(* CODESYS project tt_serialcommunication.library
   Company: Trimech Technology
   Version: 1.0
   Placeholder: TT_SerialCom_Lib
   Author: Beckhoff Singapore
   Title: TT_SerialCom_Lib

Project tree, tasks and I/O mapping:
  libraries: Tc2_SerialCom, * (Beckhoff Automation GmbH); Tc2_Standard, * (Beckhoff Automation GmbH); Tc2_System, * (Beckhoff Automation GmbH); Tc3_Module, * (Beckhoff Automation GmbH); Tc3_Interfaces, * (Beckhoff Automation GmbH)
  GVL/
    global variables TT_SerialComm_GVL
  Custom Datatypes/
    data type TT_Serial_COMBUFFER
    data type TT_Serial_FunctionResult
    data type TT_Serial_StringFormat
  Version/
    global variables Global_Version
  function block TT_Serial_StandardTask [ST]: ReadString80, SendString80
  function block TT_Serial_FastBackgroundTask [ST]: Update_Channel
  global variables TT_SerialComm_Parameters
*)

// Custom Datatypes/TT_Serial_COMBUFFER
TYPE TT_Serial_COMBUFFER :
STRUCT
(**)
	(* PLC to IO interface *)
	txBuffer 		: ComBuffer;
	rxBuffer 		: ComBuffer;
(**)
(**)	
	(* Buffers for EL COM *)
	rxElComBuffer AT %I* 	: EL6inData22B;
	txElComBuffer AT %Q* 	: EL6outData22B;
(**)
(**)
	(* Buffers for PC COM *)
	rxPcComBuffer AT %I* 	: PcComInData;
	txPcComBuffer AT %Q* 	: PcComOutData;
(**)
END_STRUCT
END_TYPE

// Custom Datatypes/TT_Serial_FunctionResult
TYPE TT_Serial_FunctionResult :
(
	NO_ERROR := -1,
	BUSY := 0,
	COM_SEND_ERROR,
	COM_RECEIVE_ERROR,
	COM_NO_STRING_RECEIVED
);
END_TYPE

// Custom Datatypes/TT_Serial_StringFormat
TYPE TT_Serial_StringFormat :
STRUCT
	Prefix : STRING;
	Surfix : STRING;
END_STRUCT
END_TYPE

// GVL/TT_SerialComm_GVL
VAR_GLOBAL
	SerialComBuffer 	: ARRAY [1..MAX_CHANNELS] OF TT_Serial_ComBuffer;
	SerialStringFormat	: ARRAY [1..MAX_CHANNELS] OF TT_Serial_StringFormat;
END_VAR

// Version/Global_Version
// This function has been automatically generated from the project information.
VAR_GLOBAL CONSTANT
	{attribute 'const_non_replaced'}
	stLibVersion_TT_SerialCom_Lib : ST_LibVersion := (iMajor := 1, iMinor := 0, iBuild := 0, iRevision := 0, sVersion := '1.0');
END_VAR

// TT_SerialComm_Parameters
VAR_GLOBAL CONSTANT
	MAX_CHANNELS 	: INT := 2;
END_VAR

// TT_Serial_StandardTask
FUNCTION_BLOCK TT_Serial_StandardTask
VAR_OUTPUT
END_VAR
VAR
	fbSendString 	: ARRAY[1..MAX_CHANNELS] OF SendString;
	fbReceiveString : ARRAY[1..MAX_CHANNELS] OF ReceiveString; (*String default 80. for 255, use ReceiveString255*)
	
	SendFlag 		: ARRAY[1..MAX_CHANNELS] OF BOOL;
	SendDataBuffer	: ARRAY[1..MAX_CHANNELS] OF STRING;
END_VAR

;

METHOD PUBLIC ReadString80 : TT_Serial_FunctionResult
VAR_INPUT
	CHANNEL 			: INT;
	RECEIVED_DATA		: POINTER TO STRING;
END_VAR
VAR 
	String_Data_Buffer 	: STRING;
END_VAR
fbReceiveString[CHANNEL](
	Prefix:= SerialStringFormat[CHANNEL].Prefix, 
	Suffix:= SerialStringFormat[CHANNEL].Surfix, 
	Timeout:= T#1S, 
	ReceivedString:= String_Data_Buffer, 
	RXbuffer:= SerialComBuffer[CHANNEL].rxBuffer );
IF fbReceiveString[CHANNEL].Error > 0 THEN
	ReadString80 := TT_Serial_FunctionResult.COM_RECEIVE_ERROR;
END_IF
IF fbReceiveString[CHANNEL].StringReceived THEN
	RECEIVED_DATA^ := String_Data_Buffer;
	ReadString80 := TT_Serial_FunctionResult.NO_ERROR;
ELSIF fbReceiveString[CHANNEL].Busy THEN
	ReadString80 := TT_Serial_FunctionResult.BUSY;
ELSE
	ReadString80 := TT_Serial_FunctionResult.COM_NO_STRING_RECEIVED;
END_IF
END_METHOD

METHOD PUBLIC SendString80 : TT_Serial_FunctionResult
VAR_INPUT
	CHANNEL	: INT;		(* The Serial Comm channel to send *)
	DATA	: STRING;	(* Without prefix & surfix *)
END_VAR
VAR
	fbTRIG 	: F_TRIG;
END_VAR
SendDataBuffer[CHANNEL] := CONCAT(SerialStringFormat[CHANNEL].Prefix, CONCAT(DATA, SerialStringFormat[CHANNEL].Surfix));
fbSendString[CHANNEL](SendString:= SendDataBuffer[CHANNEL], TXbuffer:= SerialComBuffer[CHANNEL].txBuffer);
IF fbSendString[CHANNEL].Error > 0 THEN
	SendString80 := TT_Serial_FunctionResult.COM_SEND_ERROR;
END_IF
IF fbSendString[CHANNEL].Busy THEN
	SendString80 := TT_Serial_FunctionResult.BUSY;
ELSE
	SendString80 := TT_Serial_FunctionResult.NO_ERROR;
END_IF
END_METHOD

END_FUNCTION_BLOCK

// TT_Serial_FastBackgroundTask
FUNCTION_BLOCK TT_Serial_FastBackgroundTask
VAR
	fbSerialLineControl	: ARRAY[1..MAX_CHANNELS] OF SERIALLINECONTROL;
END_VAR

;

METHOD PUBLIC Update_Channel : INT
VAR_INPUT
	CHANNEL : INT;
END_VAR
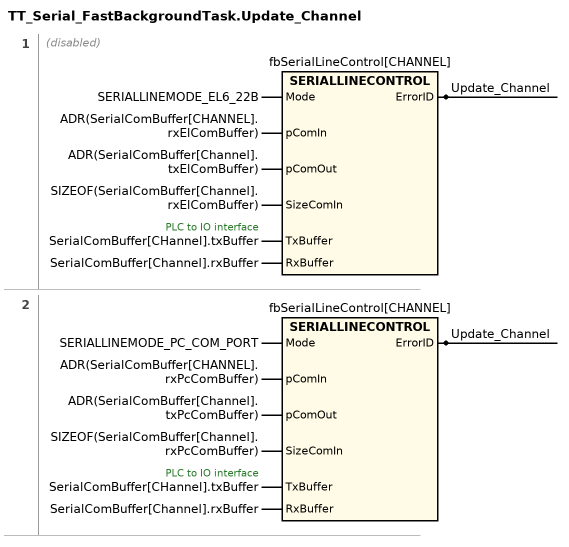
// NETWORK 1 (disabled)
//   SerialComBuffer[CHannel].txBuffer: PLC to IO interface
// fbSerialLineControl[CHANNEL](
//     Mode := SERIALLINEMODE_EL6_22B,
//     pComIn := ADR(SerialComBuffer[CHANNEL].rxElComBuffer),
//     pComOut := ADR(SerialComBuffer[Channel].txElComBuffer),
//     SizeComIn := SIZEOF(SerialComBuffer[Channel].rxElComBuffer),
//     TxBuffer := SerialComBuffer[CHannel].txBuffer,
//     RxBuffer := SerialComBuffer[Channel].rxBuffer,
//     ErrorID => Update_Channel); // SERIALLINECONTROL

// NETWORK 2
//   SerialComBuffer[CHannel].txBuffer: PLC to IO interface
fbSerialLineControl[CHANNEL](
    Mode := SERIALLINEMODE_PC_COM_PORT,
    pComIn := ADR(SerialComBuffer[CHANNEL].rxPcComBuffer),
    pComOut := ADR(SerialComBuffer[Channel].txPcComBuffer),
    SizeComIn := SIZEOF(SerialComBuffer[Channel].rxPcComBuffer),
    TxBuffer := SerialComBuffer[CHannel].txBuffer,
    RxBuffer := SerialComBuffer[Channel].rxBuffer,
    ErrorID => Update_Channel); // SERIALLINECONTROL
END_METHOD

END_FUNCTION_BLOCK
